PROGRAM HMI
VAR
	eChargerType : E_ChargerType;
	
	SysCLK					: GETSYSTEMTIME;
	//fileTime				: T_FILETIME;
	LastTimeShot			: STRING;
	ChargeGraphTMR_TON		: TON;
	ChargeGraphTMR_PT		: TIME := ChargeTime_DB.LongestChargeTime_PT + T#10S;
	ChargeGraphTMR_ET		: TIME;
	LongestChargeTIME		: REAL;
	LastTimeShotLog			: BOOL;
	
	i : INT := 1;
	n : INT := 7;

	LastTimeShotTMR_TON		: TON;
	LastTimeShotTMR_PT		: TIME := T#120H;
	LastTimeShotTMR_ET		: TIME;
	LastTimeShotTMR_REAL	: DWORD;
END_VAR

// if clear all faults, reset abort status
IF HMI_DB.ClearFaultPB = TRUE THEN
	Trips_DB.ChargedTimerRunout := FALSE;
	Trips_DB.ChargingTimerRunout := FALSE;
	Trips_DB.DumpTimerRunout := FALSE;
	Trips_DB.ChargerSummaryFault := FALSE;
	Trips_DB.ShortingSystemUnknown := FALSE;
	Trips_DB.AnyEstopPressed := FALSE;
END_IF

IF Trips_DB.ChargedTimerRunout = TRUE OR 
	Trips_DB.ChargingTimerRunout = TRUE //OR 
	//Trips_DB.DumpTimerRunout = TRUE 
	THEN
		Trips_DB.TimerRunOutON := TRUE; 
		ELSE
			Trips_DB.TimerRunOutON := FALSE;
		END_IF


LastTimeShotTMR_TON (IN := TRUE, PT := LastTimeShotTMR_PT, ET => LastTimeShotTMR_ET);

IF (Sequence.eState = E_State.CHARGECOMPLETE) AND HMI_DB.FirePB = TRUE THEN 
	//SysCLK (timeLoDW => fileTime.dwLowDateTime, timeHiDW => fileTime.dwHighDateTime);
	//LastTimeShot := SYSTEMTIME_TO_STRING( FILETIME_TO_SYSTEMTIME( fileTime ) );	
	LastTimeShotTMR_TON (IN := FALSE, PT := LastTimeShotTMR_PT, ET => LastTimeShotTMR_ET);
	HMI_DB.LastTimeShotLog := TRUE;	
	ELSE
		HMI_DB.LastTimeShotLog := FALSE;
END_IF

LastTimeShotTMR_REAL := TIME_TO_DWORD (LastTimeShotTMR_ET)/1000;

IF (Sequence.eState = E_State.CHARGECOMPLETE OR Sequence.eState = E_State.CHARGING) THEN
	ChargeGraphTMR_TON (IN:= TRUE, PT:= ChargeGraphTMR_PT, ET => ChargeGraphTMR_ET);
	ELSE
		ChargeGraphTMR_TON (IN:= FALSE);
END_IF

LongestChargeTIME := TIME_TO_REAL (ChargeGraphTMR_ET)/1000;


IF i > n THEN 
	i := 1;
END_IF

END_PROGRAM

(* stored: Version 1.1.0.1, ProductVersion 3.1.4024.11
   POU HMI: Id {dcabf1a6-3ca3-40de-943d-43b2e4fd41d0}, SpecialFunc None *)
